# EPICS substitutions: examples/test/breaktable/db/telemessEddyCurrentSensors.substitutions
file "ecmcEcSlave.template"
{
  pattern {}
          {}
}

#Actually the scalinging is between 0..10.737V (see manual)
file "ecmcEL3XXX-chX.template"
{
  pattern {CH_ID, LINR,                      ESLO, EOFF,   EGU,        PREC, LOW, LOLO,  HIGH,  HIHI,  HYST, LLSV,    LSV,     HSV,     HHSV   }
          {1,     "typeTelemess33020_21877", 1,    0,      "mm",       3,    0,   -1,    15,    16,    0,    "MAJOR", "MINOR", "MINOR", "MAJOR"}
          {2,     "typeTelemess33021_21878", 1,    0,      "mm",       3,    0,   -1,    15,    16,    0,    "MAJOR", "MINOR", "MINOR", "MAJOR"}
          {3,     "typeTelemess33018_21876", 1,    0,      "mm",       3,    0,   -1,    15,    16,    0,    "MAJOR", "MINOR", "MINOR", "MAJOR"}
          {4,     "typeTelemess32900_21875", 1,    0,      "mm",       3,    0,   -1,    20,    21,    0,    "MAJOR", "MINOR", "MINOR", "MAJOR"}
}
